TYPE ST_ScrewdriverPositionConfig :
STRUCT
    stReady : ST_Point3D;
    stWork : ST_Point3D;
END_STRUCT
END_TYPE

(* stored: Version 1.1.0.1, ProductVersion 3.1.4026.20
   DUT ST_ScrewdriverPositionConfig: Id {0cba4350-a43b-45cf-8b39-e96286d90847} *)
